// SIMATIC S7-200 project (STEP 7-Micro/WIN), CPU 221 REL 01.10

ORGANIZATION_BLOCK 主程序:OB1
TITLE=程序注释
BEGIN
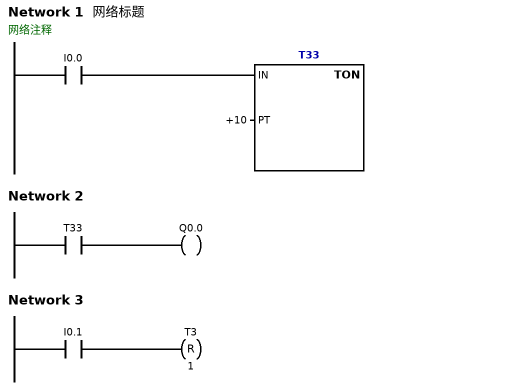
Network 1 // 网络标题
// 网络注释
LD     I0.0
TON    T33, +10
Network 2
// (network saved uncompiled; LAD cells follow)
// row 0: c0 -| |- T33  c1 -( ) Q0.0
Network 3
LD     I0.1
R      T3, 1
END_ORGANIZATION_BLOCK
